// TIA Portal V17 export
// export: Created 2022-03-29T18:52:12.1585154Z, ExportSetting WithDefaults, DisplayName Totally Integrated Automation Portal, DisplayVersion V17, DisplayName TIA Portal Openness, DisplayVersion V17, DisplayName TIA Portal Version Control Interface, DisplayVersion V17, DisplayName STEP 7 Professional, DisplayVersion V17, DisplayName STEP 7 Safety, DisplayVersion V17, DisplayName WinCC Advanced / Unified PC, DisplayVersion V17
FUNCTION_BLOCK "EM00_CM04_ConveyorCrossing"   // FB31654, LAD
TITLE = EM00_CM04
{ S7_Optimized_Access := 'TRUE' }
AUTHOR : tech.team.motioncontrol@siemens.com
FAMILY : CPG
VERSION : 1.1
// Support: tech.team.motioncontrol@siemens.com
// stored: AutoNumber true, IsIECCheckEnabled false, IsRetainMemResEnabled false, MemoryReserve 100, SetENOAutomatically false, UDAEnableTagReadback false
   VAR
      statDummyBool { ExternalAccessible := 'False'; ExternalVisible := 'False'; ExternalWritable := 'False'} : Bool;   // dummy bool - placeholder
      instConveyorCrossing { S7_SetPoint := 'True'} : "ConveyorCrossing";
   END_VAR
BEGIN

REGION Network 1: *** Begin the Setpoint Management Information Section ***
END_REGION

REGION Network 2: *** Begin the Logic Section ***
END_REGION

REGION Network 3: Conveyor crossing instance
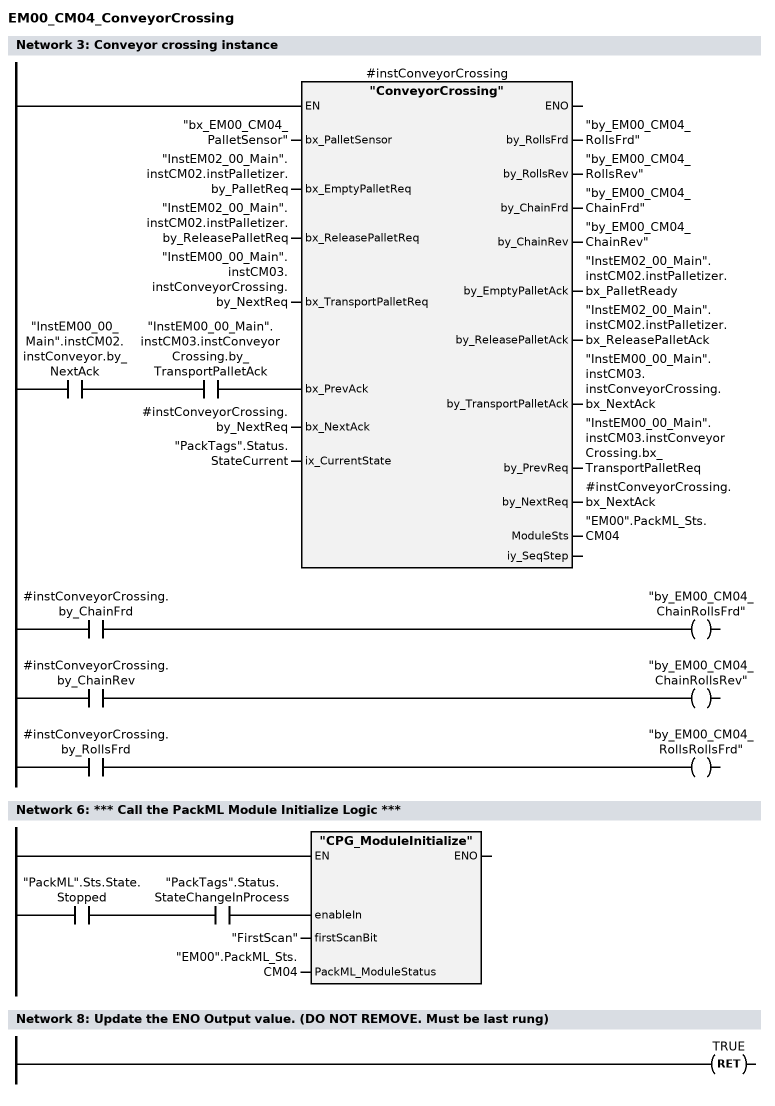
   RUNG wire#powerrail
      #instConveyorCrossing(bx_PrevAck := wire#w1, bx_PalletSensor := "bx_EM00_CM04_PalletSensor", bx_EmptyPalletReq := "InstEM02_00_Main".instCM02.instPalletizer.by_PalletReq, bx_ReleasePalletReq := "InstEM02_00_Main".instCM02.instPalletizer.by_ReleasePalletReq, bx_TransportPalletReq := "InstEM00_00_Main".instCM03.instConveyorCrossing.by_NextReq, bx_NextAck := #instConveyorCrossing.by_NextReq, ix_CurrentState := "PackTags".Status.StateCurrent, by_RollsFrd => "by_EM00_CM04_RollsFrd", by_RollsRev => "by_EM00_CM04_RollsRev", by_ChainFrd => "by_EM00_CM04_ChainFrd", by_ChainRev => "by_EM00_CM04_ChainRev", by_EmptyPalletAck => "InstEM02_00_Main".instCM02.instPalletizer.bx_PalletReady, by_ReleasePalletAck => "InstEM02_00_Main".instCM02.instPalletizer.bx_ReleasePalletAck, by_TransportPalletAck => "InstEM00_00_Main".instCM03.instConveyorCrossing.bx_NextAck, by_PrevReq => "InstEM00_00_Main".instCM03.instConveyorCrossing.bx_TransportPalletReq, by_NextReq => #instConveyorCrossing.bx_NextAck, ModuleSts => "EM00".PackML_Sts.CM04, iy_SeqStep =>)
   END_RUNG
   RUNG wire#powerrail
      Contact( "InstEM00_00_Main".instCM02.instConveyor.by_NextAck )
      Contact( "InstEM00_00_Main".instCM03.instConveyorCrossing.by_TransportPalletAck )
   END_RUNG wire#w1
   RUNG wire#powerrail
      Contact( #instConveyorCrossing.by_ChainFrd )
      Coil( "by_EM00_CM04_ChainRollsFrd" )
   END_RUNG
   RUNG wire#powerrail
      Contact( #instConveyorCrossing.by_ChainRev )
      Coil( "by_EM00_CM04_ChainRollsRev" )
   END_RUNG
   RUNG wire#powerrail
      Contact( #instConveyorCrossing.by_RollsFrd )
      Coil( "by_EM00_CM04_RollsRollsFrd" )
   END_RUNG
   // the same network as SCL:
   #instConveyorCrossing(bx_PalletSensor := "bx_EM00_CM04_PalletSensor",   // "ConveyorCrossing"
                         bx_EmptyPalletReq := "InstEM02_00_Main".instCM02.instPalletizer.by_PalletReq,
                         bx_ReleasePalletReq := "InstEM02_00_Main".instCM02.instPalletizer.by_ReleasePalletReq,
                         bx_TransportPalletReq := "InstEM00_00_Main".instCM03.instConveyorCrossing.by_NextReq,
                         bx_PrevAck := "InstEM00_00_Main".instCM02.instConveyor.by_NextAck AND "InstEM00_00_Main".instCM03.instConveyorCrossing.by_TransportPalletAck,
                         bx_NextAck := #instConveyorCrossing.by_NextReq,
                         ix_CurrentState := "PackTags".Status.StateCurrent,
                         by_RollsFrd => "by_EM00_CM04_RollsFrd",
                         by_RollsRev => "by_EM00_CM04_RollsRev",
                         by_ChainFrd => "by_EM00_CM04_ChainFrd",
                         by_ChainRev => "by_EM00_CM04_ChainRev",
                         by_EmptyPalletAck => "InstEM02_00_Main".instCM02.instPalletizer.bx_PalletReady,
                         by_ReleasePalletAck => "InstEM02_00_Main".instCM02.instPalletizer.bx_ReleasePalletAck,
                         by_TransportPalletAck => "InstEM00_00_Main".instCM03.instConveyorCrossing.bx_NextAck,
                         by_PrevReq => "InstEM00_00_Main".instCM03.instConveyorCrossing.bx_TransportPalletReq,
                         by_NextReq => #instConveyorCrossing.bx_NextAck,
                         ModuleSts => "EM00".PackML_Sts.CM04);
   "by_EM00_CM04_ChainRollsFrd" := #instConveyorCrossing.by_ChainFrd;
   "by_EM00_CM04_ChainRollsRev" := #instConveyorCrossing.by_ChainRev;
   "by_EM00_CM04_RollsRollsFrd" := #instConveyorCrossing.by_RollsFrd;
END_REGION

REGION Network 4: *** Begin the Event Information Section ***
END_REGION

REGION Network 5: *** Begin the State Model Status Feedback Section ***
END_REGION

REGION Network 6: *** Call the PackML Module Initialize Logic ***
   RUNG wire#powerrail
      "CPG_ModuleInitialize"(enableIn := wire#w1, firstScanBit := "FirstScan", PackML_ModuleStatus := "EM00".PackML_Sts.CM04)
   END_RUNG
   RUNG wire#powerrail
      Contact( "PackML".Sts.State.Stopped )
      Contact( "PackTags".Status.StateChangeInProcess )
   END_RUNG wire#w1
   // the same network as SCL:
   "CPG_ModuleInitialize"(enableIn := "PackML".Sts.State.Stopped AND "PackTags".Status.StateChangeInProcess,
                          firstScanBit := "FirstScan",
                          PackML_ModuleStatus := "EM00".PackML_Sts.CM04);
END_REGION

REGION Network 8: Update the ENO Output value. (DO NOT REMOVE. Must be last rung)
   RUNG wire#powerrail
      ReturnCoil( TRUE )
   END_RUNG
   // the same network as SCL:
   ENO := TRUE;
   RETURN;
END_REGION
END_FUNCTION_BLOCK
